FUNCTION_BLOCK FB_axisCtrl
VAR_INPUT
	
END_VAR
VAR_OUTPUT
END_VAR
VAR_IN_OUT     
	stAxisCtrl	:ST_axisCtrl; 	
	IN_OUT 		: ST_MotionAxis_MC	;//struct for each axis
END_VAR
VAR
	ton_delay	: TON;
END_VAR

//add timeout for this fuction block
ton_delay(PT:= T#2S);
CASE stAxisCtrl.iCmd OF
	0:
		IN_OUT.mcReset.Execute	:= FALSE;
		IN_OUT.mcStop.Execute	:= FALSE	;
	1:
		IN_OUT.mcPower.Enable	:= TRUE;
		stAxisCtrl.iCmd	:= 0;
	2:
		IN_OUT.mcPower.Enable	:= FALSE;
		stAxisCtrl.iCmd	:= 0;	
	3:
		IN_OUT.mcReset.Execute	:= TRUE;
		stAxisCtrl.iCmd	:= 0;
	4:
		IN_OUT.mcStop.Execute	:= TRUE;
		stAxisCtrl.iCmd	:= 0;	
	5: 
		IN_OUT.mcMoveAbsolute.Execute := TRUE;
		IN_OUT.rActualPosSet	:= stAxisCtrl.rPosition;
		IN_OUT.rVelocitySet	:= stAxisCtrl.iSpeed;
		IF IN_OUT.mcMoveAbsolute.Done THEN
			stAxisCtrl.iCmd	:= 0;
		END_IF
		
	10://REM aging test start
		ton_delay.IN	:= FALSE;
		IN_OUT.mcMoveAbsolute.Execute := TRUE;
		IN_OUT.rActualPosSet	:= 0;
		IN_OUT.rVelocitySet	:= 100;
		IF IN_OUT.mcMoveAbsolute.Done THEN
			IN_OUT.mcMoveAbsolute.Execute := FALSE;
			stAxisCtrl.iCmd	:= 11;
		END_IF
	11:
		ton_delay.IN	:= TRUE;
		IF ton_delay.Q THEN
			stAxisCtrl.iCmd	:= 12;
		END_IF
	12:
		ton_delay.IN	:= FALSE;
		IN_OUT.mcMoveAbsolute.Execute := TRUE;
		IN_OUT.rActualPosSet	:= 0;
		IN_OUT.rVelocitySet	:= 100;
		IF IN_OUT.mcMoveAbsolute.Done THEN
			IN_OUT.mcMoveAbsolute.Execute := FALSE;
			stAxisCtrl.iCmd	:= 13;
		END_IF
	13:
		ton_delay.IN	:= TRUE;
		IF ton_delay.Q THEN
			stAxisCtrl.iCmd	:= 10;
		END_IF	
	
		
	20://PM buffer aging test start
		IN_OUT.mcSetpoint.Execute	:= 0;
		stAxisCtrl.iCmd	:= 21;
	21:
		IN_OUT.mcMoveVelocity.Execute	:= TRUE;
		IN_OUT.rVelocity	:= 100;
		
	
	
	
	
	100:
		IN_OUT.mcMoveAbsolute.Execute := FALSE;
		IN_OUT.mcMoveVelocity.Execute	:= FALSE;
		IN_OUT.mcStop.Execute	:= TRUE;
		stAxisCtrl.iCmd	:= 0;
		
END_CASE;
stAxisCtrl.iStatus := stAxisCtrl.iCmd;

END_FUNCTION_BLOCK

(* stored: Version 1.1.0.1, ProductVersion 3.1.4024.12
   POU FB_axisCtrl: Id {2ac385ec-b262-4b8e-ba8d-e1a3f0cb06b1}, SpecialFunc None *)
